(* IEC 61131-3 sources: SmartHomeNew/snapshots/project_clean_state_2026_04_16, 22 files *)

(* ---- CONSTANTS.dut ---- *)
TYPE
    C_MAX_HEATING_CIRCUITS : INT := 8;
    C_MAX_LIGHTING_ZONES : INT := 32;
    C_MAX_CLIMATE_ZONES : INT := 16;
    C_MAX_VENT_UNITS : INT := 8;
    C_MAX_DHW_UNITS : INT := 4;
    C_MAX_IO_MODULES : INT := 16;
END_TYPE

(* ---- ST_Blinds_Command_V2.dut ---- *)
TYPE ST_Blinds_Command_V2 :
STRUCT
    Position_Setpoint : BYTE;
END_STRUCT
END_TYPE

(* ---- ST_Blinds_State_V2.dut ---- *)
TYPE ST_Blinds_State_V2 :
STRUCT
    Position_Actual : BYTE;
END_STRUCT
END_TYPE

(* ---- ST_Debug_Logger_Config.dut ---- *)
{attribute 'pack_mode' := '1'}
TYPE ST_Debug_Logger_Config :
STRUCT
    enabled : BOOL;
    sampling_period_ms : UDINT := GVL_CONSTANTS.C_MS_IN_SECOND;
END_STRUCT
END_TYPE

(* ---- ST_DHW_Command_V2.dut ---- *)
TYPE ST_DHW_Command_V2 :
STRUCT
    Pump_Enable : REAL;
END_STRUCT
END_TYPE

(* ---- ST_Lifetime_Status.dut ---- *)
{attribute 'pack_mode' := '1'}
TYPE ST_Lifetime_Status :
STRUCT
    device_id : BYTE;
    runtime_hours : UDINT;
    start_count : UDINT;
    remaining_hours : UDINT;
    remaining_percent : BYTE;
    maintenance_required : BOOL;
    last_calc_timestamp : UDINT;
END_STRUCT
END_TYPE

(* ---- ST_Trend_History_Record.dut ---- *)
{attribute 'pack_mode' := '1'}
TYPE ST_Trend_History_Record :
STRUCT
    timestamp_ms : UDINT := 0;
    value : REAL := 0.0;
END_STRUCT
END_TYPE

(* ---- ST_Ventilation_State_V2.dut ---- *)
TYPE ST_Ventilation_State_V2 : STRUCT
    Supply_Temp : REAL;
END_STRUCT
END_TYPE

(* ---- FB_DHW_V2_Staging.st ---- *)
FUNCTION_BLOCK FB_DHW_V2_Staging
VAR_INPUT
    VI_Tank_ID : INT;
    VI_Enable : BOOL;
    VI_Target_Temp : REAL;
    VI_Pump_Enable : BOOL;
    VI_Heating_Priority : BOOL;
    VI_Is_Active : BOOL;
    VI_Tank_Temp : REAL;
    VI_Supply_Temp : REAL;
    VI_Return_Temp : REAL;
    VI_Pump_Actual : BOOL;
    VI_Alarm_Active : BOOL;
END_VAR
VAR_OUTPUT
    VO_Command_Shadow : ST_DHW_Command_V2;
    VO_State_Shadow : ST_DHW_State_V2;
END_VAR

IF VI_Pump_Enable THEN
    VO_Command_Shadow.Pump_Enable := 1.0;
ELSE
    VO_Command_Shadow.Pump_Enable := 0.0;
END_IF;

VO_State_Shadow.Tank_Temp := VI_Tank_Temp;
VO_State_Shadow.Supply_Temp := VI_Supply_Temp;
END_FUNCTION_BLOCK

(* ---- FB_NVRAM_Manager.st ---- *)
FUNCTION_BLOCK FB_NVRAM_Manager
VAR_INPUT
    VI_Command                  : BYTE; // 1=WRITE, 2=READ
    VI_Offset                   : UDINT; // Смещение в байтах
    VI_DataRef                  : REFERENCE TO BYTE;
    VI_DataSize                 : UDINT; // КРИТИЧНО: используем этот размер вместо SIZEOF
    VI_System_Time_MS           : UDINT;
    VI_Operator_ID              : STRING(10);
    VI_IsActivePLC              : BOOL;
    VI_TwoPersonConfirmation    : BOOL;
END_VAR
VAR_OUTPUT
    VO_Done                     : BOOL;
    VO_Error                    : BOOL;
    VO_ErrorID                  : UDINT;
    // VO_ReadDataRef removed (REFERENCE TO not allowed in output)
    VO_HMI_Status_Message       : STRING(200);
END_VAR
VAR
    L_prev_Command              : BYTE;
    L_cmd_rising                : BOOL;
    L_i                         : UDINT;
    L_Last_Write_Time_MS        : UDINT := 0; // Время последней записи
    L_Data_Changed              : BOOL; // Флаг изменения данных
    L_pData                      : POINTER TO BYTE;
END_VAR
VAR CONSTANT
    C_MAX_NVRAM_SIZE            : UDINT := 12800;
END_VAR

// Детекция фронта команды
L_cmd_rising := (VI_Command <> 0) AND (L_prev_Command = 0);
L_prev_Command := VI_Command;

IF L_cmd_rising THEN
    VO_Done := FALSE;
    VO_Error := FALSE;
    VO_ErrorID := 0;
    VO_HMI_Status_Message := '';

    // Валидация смещения
    IF VI_Offset >= C_MAX_NVRAM_SIZE THEN
        VO_Error := TRUE;
        VO_ErrorID := 16#1501;
        VO_HMI_Status_Message := 'NVRAM: Неверное смещение';
        VO_Done := TRUE;
        RETURN;
    END_IF;

    // Валидация указателя
    IF NOT __ISVALIDREF(VI_DataRef) THEN
        VO_Error := TRUE;
        VO_ErrorID := 16#150A;
        VO_HMI_Status_Message := 'NVRAM: Недействительная ссылка на данные';
        VO_Done := TRUE;
        RETURN;
    END_IF;

    L_pData := ADR(VI_DataRef);

    IF (VI_Offset + VI_DataSize) > C_MAX_NVRAM_SIZE THEN
        VO_Error := TRUE;
        VO_ErrorID := 16#150B;
        VO_HMI_Status_Message := 'NVRAM: Размер данных превышает доступный объем';
        VO_Done := TRUE;
        RETURN;
    END_IF;

    IF VI_Command = 1 THEN // ЗАПИСЬ (WRITE)
        IF NOT VI_IsActivePLC THEN
            VO_Error := TRUE;
            VO_ErrorID := 16#1509;
            VO_HMI_Status_Message := 'NVRAM: Запись запрещена (STANDBY)';
        ELSE
            // Ограничение частоты записи (не чаще 1 раза в 60 секунд)
            IF (VI_System_Time_MS - L_Last_Write_Time_MS) < 60000 AND L_Last_Write_Time_MS <> 0 THEN
                VO_Error := TRUE;
                VO_ErrorID := 16#150C;
                VO_HMI_Status_Message := 'NVRAM: Превышена частота записи (лимит 1 раз в 60с)';
            ELSE
                // Проверка на изменение данных перед записью
                L_Data_Changed := FALSE;
                IF TRUE THEN
                    L_Data_Changed := TRUE;
                END_IF;

                IF L_Data_Changed THEN
                    // Безопасное копирование (WRITE)
                    FOR L_i := 0 TO VI_DataSize - 1 DO
                        GVL_Retain.G_NVRAM_Data[VI_Offset + L_i] := L_pData[L_i];
                    END_FOR;
                    L_Last_Write_Time_MS := VI_System_Time_MS;
                    VO_HMI_Status_Message := 'NVRAM: Данные успешно сохранены в RETAIN';
                ELSE
                    VO_HMI_Status_Message := 'NVRAM: Данные не изменились, запись пропущена';
                END_IF;
            END_IF;
        END_IF;
        VO_Done := TRUE;

    ELSIF VI_Command = 2 THEN // ЧТЕНИЕ (READ)
        // Безопасное копирование (READ)
        FOR L_i := 0 TO VI_DataSize - 1 DO
            L_pData[L_i] := GVL_Retain.G_NVRAM_Data[VI_Offset + L_i];
        END_FOR;
        VO_HMI_Status_Message := 'NVRAM: Данные успешно прочитаны из RETAIN';
        VO_Done := TRUE;
    END_IF;
END_IF;

IF VI_Command = 0 THEN
    VO_Done := FALSE;
END_IF;
// >>> BULK_SYNC_ANCHOR: FB_NVRAM_Manager <<<

(* ---- FB_PID_Controller.st ---- *)
FUNCTION_BLOCK FB_PID_Controller
VAR_INPUT
    VI_SetPoint : REAL;         // Уставка
    VI_ProcessValue : REAL;     // Текущее значение
    VI_Kp : REAL;               // Коэффициент усиления
    VI_Tn : REAL;               // Время интегрирования (сек)
    VI_Tv : REAL;               // Время дифференцирования (сек)
    VI_Y_Min : REAL := 0.0;     // Минимальный выход
    VI_Y_Max : REAL := 100.0;   // Максимальный выход
    VI_Manual_Mode : BOOL;      // Ручной режим
    VI_Manual_Value : REAL;     // Значение в ручном режиме
    VI_Deadband : REAL := 0.1;  // Мертвая зона
    VI_Cycle_Time_S : REAL := 0.01; // Время цикла задачи в секундах
    VI_Reset : BOOL;            // Сброс интегральной составляющей
END_VAR
VAR_OUTPUT
    VO_Output : REAL;           // Выход регулятора
    VO_Error : REAL;            // Ошибка рассогласования
    VO_Limiting : BOOL;         // Флаг ограничения выхода (Anti-windup)
END_VAR
VAR
    L_Integral_Sum : REAL;      // Интегральная сумма
    L_Prev_Error : REAL;        // Предыдущая ошибка
    L_Derivative : REAL;        // Дифференциальная составляющая
    L_Output_Raw : REAL;        // Сырой выход до ограничения
END_VAR

// Расчет ошибки
VO_Error := VI_SetPoint - VI_ProcessValue;

// Проверка мертвой зоны
IF ABS(VO_Error) < VI_Deadband THEN
    VO_Error := 0.0;
END_IF;

IF VI_Reset THEN
    L_Integral_Sum := 0.0;
    L_Prev_Error := 0.0;
    VO_Output := 0.0;
    RETURN;
END_IF;

IF VI_Manual_Mode THEN
    VO_Output := VI_Manual_Value;
    // Безударный переход: при выходе из ручного режима выход должен остаться прежним.
    // Так как Выход = P + I + D, то I = Выход - P - D.
    // Для простоты D при переходе обнуляем (или игнорируем), тогда I = Выход - P.
    L_Integral_Sum := VO_Output - (VI_Kp * VO_Error);
    L_Prev_Error := VO_Error;
    RETURN;
END_IF;

// Пропорциональная составляющая
L_Output_Raw := VI_Kp * VO_Error;

// Интегральная составляющая (Метод трапеций)
IF VI_Tn > 0.0 THEN
    // Anti-windup: не накапливаем интеграл, если выход уже на пределе и ошибка того же знака
    IF NOT VO_Limiting OR (VO_Error > 0.0 AND L_Output_Raw < VI_Y_Max) OR (VO_Error < 0.0 AND L_Output_Raw > VI_Y_Min) THEN
        L_Integral_Sum := L_Integral_Sum + (VI_Kp / VI_Tn) * VO_Error * VI_Cycle_Time_S;
    END_IF;
    L_Output_Raw := L_Output_Raw + L_Integral_Sum;
END_IF;

// Дифференциальная составляющая
IF VI_Tv > 0.0 THEN
    L_Derivative := (VO_Error - L_Prev_Error) / VI_Cycle_Time_S;
    L_Output_Raw := L_Output_Raw + VI_Kp * VI_Tv * L_Derivative;
END_IF;

L_Prev_Error := VO_Error;

// Ограничение выхода
IF L_Output_Raw > VI_Y_Max THEN
    VO_Output := VI_Y_Max;
    VO_Limiting := TRUE;
ELSIF L_Output_Raw < VI_Y_Min THEN
    VO_Output := VI_Y_Min;
    VO_Limiting := TRUE;
ELSE
    VO_Output := L_Output_Raw;
    VO_Limiting := FALSE;
END_IF;
// >>> BULK_SYNC_ANCHOR: FB_PID_Controller <<<

(* ---- FB_Pre_Departure_Heating.st ---- *)
FUNCTION_BLOCK FB_Pre_Departure_Heating
VAR_INPUT
    VI_Departure_Time : UDINT;
    VI_System_Time    : UDINT;
END_VAR
VAR_IN_OUT
    VI_Selected       : ARRAY[1..GVL_CONSTANTS.C_MAX_HEATING_CIRCUITS] OF BOOL;
END_VAR
VAR_OUTPUT
    VO_Heating_Active : BOOL;
    VO_Setpoints      : ARRAY[1..GVL_CONSTANTS.C_MAX_HEATING_CIRCUITS] OF REAL;
END_VAR

VAR
    L_i : INT;
END_VAR

// Запуск за 3 часа (10800000 мс)
IF (SEL(VI_Departure_Time >= VI_System_Time, VI_Departure_Time - VI_System_Time, (4294967295 - VI_System_Time) + VI_Departure_Time + 1)) < 10800000 THEN
    VO_Heating_Active := TRUE;
    FOR L_i := 1 TO GVL_CONSTANTS.C_MAX_HEATING_CIRCUITS DO
        IF VI_Selected[L_i] THEN VO_Setpoints[L_i] := 22.0; END_IF;
    END_FOR;
ELSE
    VO_Heating_Active := FALSE;
END_IF;

(* ---- FB_Presence_Playback.st ---- *)
FUNCTION_BLOCK FB_Presence_Playback
VAR_INPUT
    VI_Mode_Record : BOOL; // TRUE - записываем, FALSE - воспроизводим
    VI_Time_Index   : UDINT; // Индекс времени в рамках недели (мс)
END_VAR
VAR_IN_OUT
    VI_Light_Inputs : ARRAY[1..32] OF BOOL;
END_VAR
VAR_OUTPUT
    VO_Light_Outputs : ARRAY[1..32] OF BOOL;
END_VAR
VAR
    L_Current_Slot : UDINT;
    L_i : INT;
END_VAR

L_Current_Slot := (VI_Time_Index / (GVL_CONSTANTS.C_MS_IN_MINUTE * 10)) MOD TO_UDINT(GVL_CONSTANTS.C_MAX_PRESENCE_HISTORY); // Слот каждые 10 минут

IF VI_Mode_Record THEN
    // Запись текущего состояния в слот
    GVL_Retain.G_Presence_History[L_Current_Slot] := 0;
    FOR L_i := 1 TO 32 DO
        IF VI_Light_Inputs[L_i] THEN
            GVL_Retain.G_Presence_History[L_Current_Slot] := GVL_Retain.G_Presence_History[L_Current_Slot] OR SHL(WORD#1, L_i-1);
        END_IF;
    END_FOR;
ELSE
    // Воспроизведение из слота
    FOR L_i := 1 TO 32 DO
        VO_Light_Outputs[L_i] := (GVL_Retain.G_Presence_History[L_Current_Slot] AND SHL(WORD#1, L_i-1)) <> 0;
    END_FOR;
END_IF;

(* ---- FB_Redundancy_Manager.st ---- *)
FUNCTION_BLOCK FB_Redundancy_Manager
VAR_INPUT
    VI_System_Time_MS : UDINT; // Системное время (мс)
    VI_Local_PLC_ID : BYTE; // 1 = ПЛК А, 2 = ПЛК B
    VI_Remote_Pulse : BOOL; // Сигнал от партнера
    VI_Remote_Is_Active : BOOL; // Статус партнера
    VI_Gateway_Ping_OK : BOOL; // Пинг до шлюза
    VI_Remote_State : ST_System_State_Snapshot; // Состояние партнера
    VI_Local_State : ST_System_State_Snapshot; // Локальное состояние
END_VAR
VAR_OUTPUT
    VO_Local_Role : E_PLC_ROLE; // Локальная роль ПЛК (Active/Standby)
    VO_Local_Pulse : BOOL; // Локальный сигнал пульса для партнера
    VO_Sync_Data_Req : BOOL; // Запрос на синхронизацию данных
    VO_Status_Msg : STRING(200); // Строковое сообщение о статусе
    VO_Synced_State : ST_System_State_Snapshot; // Синхронизированное состояние
    VO_State_Updated : BOOL; // Флаг: Состояние было обновлено
END_VAR
VAR
    L_Heartbeat : FB_PLC_Heartbeat;
    L_Pulse_Timer : FB_System_Timer;
    L_Pulse_State : BOOL;
    L_Prev_Role : E_PLC_ROLE;
    L_State_Replicator : FB_State_Replication;
END_VAR

// 1. Генерация собственного пульса (меандр 100 мс)
L_Pulse_Timer(IN := NOT L_Pulse_Timer.Q, PT := T#100ms, VI_System_Time_MS := VI_System_Time_MS);
IF L_Pulse_Timer.Q THEN
    L_Pulse_State := NOT L_Pulse_State;
END_IF;
VO_Local_Pulse := L_Pulse_State;

// 2. Определение роли через Heartbeat
L_Heartbeat(
    VI_Local_ID := VI_Local_PLC_ID,
    VI_System_Time := VI_System_Time_MS,
    VI_Remote_Pulse := VI_Remote_Pulse,
    VI_Remote_Is_Active := VI_Remote_Is_Active,
    VI_Gateway_Ping_OK := VI_Gateway_Ping_OK
);

IF L_Heartbeat.VO_Is_Active THEN
    VO_Local_Role := E_PLC_ROLE.ROLE_ACTIVE;
    VO_Status_Msg := 'ПЛК АКТИВЕН (ВЕДУЩИЙ)';
ELSE
    VO_Local_Role := E_PLC_ROLE.ROLE_STANDBY;
    VO_Status_Msg := 'ПЛК В РЕЗЕРВЕ (ВЕДОМЫЙ)';
END_IF;

// 3. Запрос на синхронизацию при переходе в ACTIVE
IF VO_Local_Role = E_PLC_ROLE.ROLE_ACTIVE AND L_Prev_Role = E_PLC_ROLE.ROLE_STANDBY THEN
    VO_Sync_Data_Req := TRUE;
ELSE
    VO_Sync_Data_Req := FALSE;
END_IF;

L_State_Replicator(
    VI_Local_Role := VO_Local_Role,
    VI_Sync_Req := VO_Sync_Data_Req,
    VI_Local_State := VI_Local_State,
    VI_Remote_State := VI_Remote_State,
    VI_System_Time_MS := VI_System_Time_MS
);
VO_Synced_State := L_State_Replicator.VO_Synced_State;
VO_State_Updated := L_State_Replicator.VO_State_Updated;

L_Prev_Role := VO_Local_Role;
// >>> BULK_SYNC_ANCHOR: FB_Redundancy_Manager <<<

(* ---- FB_Rule_Engine.st ---- *)
FUNCTION_BLOCK FB_Rule_Engine
VAR_INPUT
    VI_System_Time_MS : UDINT; // Системное время (мс)
    VI_IsActivePLC : BOOL; // Флаг: Данный ПЛК является ведущим
    VI_Security_Armed : BOOL; // Статус: Система под охраной
    VI_Current_Time : TOD; // Текущее время суток
    VI_Day_Of_Week : INT; // Текущий день недели (1..7, 1 = Понедельник)
END_VAR
VAR_IN_OUT
    VI_Rules : ARRAY[1..GVL_CONSTANTS.C_MAX_RULES] OF ST_User_Rule; // Массив пользовательских правил
    VI_Indoor_Temps : ARRAY[1..16] OF REAL; // Температуры в помещениях
    VI_Floor_Temps : ARRAY[1..8] OF REAL; // Температуры пола
    VI_Humidities : ARRAY[1..16] OF REAL; // Влажность в помещениях
    VI_CO2_Levels : ARRAY[1..16] OF REAL; // Уровни CO2
    VI_Motion_Sensors : ARRAY[1..16] OF BOOL; // Датчики движения
    VI_Door_Sensors : ARRAY[1..GVL_CONSTANTS.C_MAX_DOOR_SENSORS] OF BOOL; // Датчики открытия дверей
    VI_Window_Sensors : ARRAY[1..16] OF BOOL; // Датчики открытия окон
    VI_Water_Sensors : ARRAY[1..GVL_CONSTANTS.C_MAX_FLOOD_SENSORS] OF BOOL; // Датчики протечки воды
    VI_Smoke_Sensors : ARRAY[1..GVL_CONSTANTS.C_MAX_SMOKE_SENSORS] OF BOOL; // Датчики дыма
    VI_Methane_Sensors : ARRAY[1..GVL_CONSTANTS.C_MAX_METHANE_SENSORS] OF REAL; // Датчики метана
    VI_CO_Sensors : ARRAY[1..GVL_CONSTANTS.C_MAX_CO_SENSORS] OF REAL; // Датчики угарного газа
END_VAR
VAR_OUTPUT
    VO_Actions : ARRAY[1..GVL_CONSTANTS.C_MAX_RULES] OF ST_Rule_Action; // Сформированные действия по правилам
END_VAR
VAR
    L_i : INT;
    fbCompat : ARRAY[1..GVL_CONSTANTS.C_MAX_RULES] OF FB_Rule_Compatibility_Package;
    L_Compat_All_OK : BOOL;
    L_Compat_First_Warning : STRING(255);
    L_Compat_First_Warning_Latched : BOOL;
    L_Shadow_V2_Enabled : BOOL;
    L_Shadow_V2_Roundtrip_Mismatch : BOOL;
    L_Shadow_V2_First_Mismatch_Rule : INT;
    L_V2_Switch_Enabled : BOOL;
    L_V2_Path_Ready : BOOL;
    L_V2_Using_Legacy_Fallback : BOOL;
    L_Condition_Met : BOOL;
    L_Current_Value : REAL;
    L_Triggers : ARRAY[1..GVL_CONSTANTS.C_MAX_RULES] OF R_TRIG;
    L_Trigger_Count : ARRAY[1..GVL_CONSTANTS.C_MAX_RULES] OF UINT;
    L_Last_Reset_Time : UDINT;
    L_Elapsed_Time : UDINT;
END_VAR

IF NOT VI_IsActivePLC THEN RETURN; END_IF;

L_Compat_All_OK := TRUE;
L_Compat_First_Warning := '';
L_Compat_First_Warning_Latched := FALSE;
L_Shadow_V2_Enabled := TRUE;
L_Shadow_V2_Roundtrip_Mismatch := FALSE;
L_Shadow_V2_First_Mismatch_Rule := 0;
L_V2_Switch_Enabled := FALSE;
L_V2_Path_Ready := FALSE;
L_V2_Using_Legacy_Fallback := TRUE;

// Сброс счетчиков срабатываний каждую минуту (защита от циклических зависимостей/дребезга)
L_Elapsed_Time := (SEL(VI_System_Time_MS >= L_Last_Reset_Time, VI_System_Time_MS - L_Last_Reset_Time, (4294967295 - L_Last_Reset_Time) + VI_System_Time_MS + 1));

IF L_Elapsed_Time >= GVL_CONSTANTS.C_MS_IN_MINUTE THEN
    L_Last_Reset_Time := VI_System_Time_MS;
    FOR L_i := 1 TO GVL_CONSTANTS.C_MAX_RULES DO
        L_Trigger_Count[L_i] := 0;
    END_FOR;
END_IF;

FOR L_i := 1 TO GVL_CONSTANTS.C_MAX_RULES DO
    fbCompat[L_i](VI_Rule_Legacy := VI_Rules[L_i]);

    IF NOT fbCompat[L_i].VO_Forward_OK OR NOT fbCompat[L_i].VO_Reverse_OK THEN
        L_Compat_All_OK := FALSE;
    END_IF;

    IF (NOT L_Compat_First_Warning_Latched) AND (fbCompat[L_i].VO_Warning_Text <> '') THEN
        L_Compat_First_Warning := fbCompat[L_i].VO_Warning_Text;
        L_Compat_First_Warning_Latched := TRUE;
    END_IF;

    IF L_Shadow_V2_Enabled THEN
        IF (fbCompat[L_i].VO_Rule_Legacy_Roundtrip.Action_Type <> VI_Rules[L_i].Action_Type)
           OR (fbCompat[L_i].VO_Rule_Legacy_Roundtrip.Action_Target_ID <> VI_Rules[L_i].Action_Target_ID)
           OR (ABS(fbCompat[L_i].VO_Rule_Legacy_Roundtrip.Action_Value - VI_Rules[L_i].Action_Value) > 0.0001)
           OR (fbCompat[L_i].VO_Rule_Legacy_Roundtrip.Condition_Type <> VI_Rules[L_i].Condition_Type)
           OR (fbCompat[L_i].VO_Rule_Legacy_Roundtrip.Condition_Target_ID <> VI_Rules[L_i].Condition_Target_ID)
           OR (fbCompat[L_i].VO_Rule_Legacy_Roundtrip.Condition_Op <> VI_Rules[L_i].Condition_Op)
           OR (ABS(fbCompat[L_i].VO_Rule_Legacy_Roundtrip.Condition_Value - VI_Rules[L_i].Condition_Value) > 0.0001)
           OR (ABS(fbCompat[L_i].VO_Rule_Legacy_Roundtrip.Condition_Value_Max - VI_Rules[L_i].Condition_Value_Max) > 0.0001) THEN
            L_Shadow_V2_Roundtrip_Mismatch := TRUE;
            IF L_Shadow_V2_First_Mismatch_Rule = 0 THEN
                L_Shadow_V2_First_Mismatch_Rule := L_i;
            END_IF;
        END_IF;
    END_IF;

    // Phase 4 scaffold: optional V2 switch point.
    // Current state: always remain on legacy behavior.
    // Future state: when V2 path is implemented and validated,
    // this block becomes the controlled branch point.
    IF L_V2_Switch_Enabled AND L_V2_Path_Ready THEN
        L_V2_Using_Legacy_Fallback := FALSE;
        // V2 action-generation path placeholder.
        // No runtime behavior change yet.
    ELSE
        L_V2_Using_Legacy_Fallback := TRUE;
    END_IF;

    VO_Actions[L_i].Active := FALSE;
    IF VI_Rules[L_i].Enabled THEN
        L_Condition_Met := FALSE;
        L_Current_Value := 0.0;

        // Определение значения для проверки
        IF VI_Rules[L_i].Condition_Target_ID > 0 THEN
            CASE VI_Rules[L_i].Condition_Type OF
                E_Rule_Condition_Type.COND_AIR_TEMP: IF VI_Rules[L_i].Condition_Target_ID <= 16 THEN L_Current_Value := VI_Indoor_Temps[VI_Rules[L_i].Condition_Target_ID]; END_IF;
                E_Rule_Condition_Type.COND_FLOOR_TEMP: IF VI_Rules[L_i].Condition_Target_ID <= 8 THEN L_Current_Value := VI_Floor_Temps[VI_Rules[L_i].Condition_Target_ID]; END_IF;
                E_Rule_Condition_Type.COND_HUMIDITY: IF VI_Rules[L_i].Condition_Target_ID <= 16 THEN L_Current_Value := VI_Humidities[VI_Rules[L_i].Condition_Target_ID]; END_IF;
                E_Rule_Condition_Type.COND_CO2: IF VI_Rules[L_i].Condition_Target_ID <= 16 THEN L_Current_Value := VI_CO2_Levels[VI_Rules[L_i].Condition_Target_ID]; END_IF;
                E_Rule_Condition_Type.COND_MOTION: IF VI_Rules[L_i].Condition_Target_ID <= 16 THEN L_Current_Value := SEL(VI_Motion_Sensors[VI_Rules[L_i].Condition_Target_ID], 0.0, 1.0); END_IF;
                E_Rule_Condition_Type.COND_DOOR_WINDOW:
                    IF VI_Rules[L_i].Condition_Target_ID <= GVL_CONSTANTS.C_MAX_DOOR_SENSORS THEN
                        L_Current_Value := SEL(VI_Door_Sensors[VI_Rules[L_i].Condition_Target_ID] OR VI_Window_Sensors[VI_Rules[L_i].Condition_Target_ID], 0.0, 1.0);
                    ELSIF VI_Rules[L_i].Condition_Target_ID <= 16 THEN
                        L_Current_Value := SEL(VI_Window_Sensors[VI_Rules[L_i].Condition_Target_ID], 0.0, 1.0);
                    END_IF;
                E_Rule_Condition_Type.COND_FLOOD: IF VI_Rules[L_i].Condition_Target_ID <= GVL_CONSTANTS.C_MAX_FLOOD_SENSORS THEN L_Current_Value := SEL(VI_Water_Sensors[VI_Rules[L_i].Condition_Target_ID], 0.0, 1.0); END_IF;
                E_Rule_Condition_Type.COND_SMOKE: IF VI_Rules[L_i].Condition_Target_ID <= GVL_CONSTANTS.C_MAX_SMOKE_SENSORS THEN L_Current_Value := SEL(VI_Smoke_Sensors[VI_Rules[L_i].Condition_Target_ID], 0.0, 1.0); END_IF;
                E_Rule_Condition_Type.COND_METHANE: IF VI_Rules[L_i].Condition_Target_ID <= GVL_CONSTANTS.C_MAX_METHANE_SENSORS THEN L_Current_Value := VI_Methane_Sensors[VI_Rules[L_i].Condition_Target_ID]; END_IF;
                E_Rule_Condition_Type.COND_CO: IF VI_Rules[L_i].Condition_Target_ID <= GVL_CONSTANTS.C_MAX_CO_SENSORS THEN L_Current_Value := VI_CO_Sensors[VI_Rules[L_i].Condition_Target_ID]; END_IF;
                E_Rule_Condition_Type.COND_TIME_OF_DAY: L_Current_Value := TO_REAL(TOD_TO_UDINT(VI_Current_Time) / GVL_CONSTANTS.C_MS_IN_MINUTE); // Время в минутах
                E_Rule_Condition_Type.COND_DAY_OF_WEEK: L_Current_Value := TO_REAL(VI_Day_Of_Week);
            END_CASE;
        ELSE
            IF VI_Rules[L_i].Condition_Type = E_Rule_Condition_Type.COND_TIME_OF_DAY THEN
                L_Current_Value := TO_REAL(TOD_TO_UDINT(VI_Current_Time) / GVL_CONSTANTS.C_MS_IN_MINUTE); // Время в минутах
            ELSIF VI_Rules[L_i].Condition_Type = E_Rule_Condition_Type.COND_DAY_OF_WEEK THEN
                L_Current_Value := TO_REAL(VI_Day_Of_Week);
            END_IF;
        END_IF;

        // Проверка условия
        CASE VI_Rules[L_i].Condition_Op OF
            E_Rule_Comparison.COMP_GT: L_Condition_Met := (L_Current_Value > VI_Rules[L_i].Condition_Value);
            E_Rule_Comparison.COMP_LT: L_Condition_Met := (L_Current_Value < VI_Rules[L_i].Condition_Value);
            E_Rule_Comparison.COMP_EQ: L_Condition_Met := (ABS(L_Current_Value - VI_Rules[L_i].Condition_Value) < 0.1);
            E_Rule_Comparison.COMP_GE: L_Condition_Met := (L_Current_Value >= VI_Rules[L_i].Condition_Value);
            E_Rule_Comparison.COMP_LE: L_Condition_Met := (L_Current_Value <= VI_Rules[L_i].Condition_Value);
            E_Rule_Comparison.COMP_IN_RANGE: L_Condition_Met := (L_Current_Value >= VI_Rules[L_i].Condition_Value) AND (L_Current_Value <= VI_Rules[L_i].Condition_Value_Max);
            E_Rule_Comparison.COMP_TRUE: L_Condition_Met := (L_Current_Value > 0.5);
            E_Rule_Comparison.COMP_FALSE: L_Condition_Met := (L_Current_Value < 0.5);
        END_CASE;

        // Формирование действия
        L_Triggers[L_i](CLK := L_Condition_Met);

        IF L_Triggers[L_i].Q THEN
            L_Trigger_Count[L_i] := L_Trigger_Count[L_i] + 1;
            IF L_Trigger_Count[L_i] > 10 THEN
                // ТЗ 13.5: Блокировка правила при слишком частом срабатывании (циклическая зависимость)
                VO_Actions[L_i].Active := FALSE;
                VO_Actions[L_i].Triggered := FALSE;
                CONTINUE; // Пропускаем выполнение
            END_IF;
        END_IF;

        IF L_Condition_Met AND (L_Trigger_Count[L_i] <= 10) THEN
            VO_Actions[L_i].Active := TRUE;
            VO_Actions[L_i].Triggered := L_Triggers[L_i].Q;
            VO_Actions[L_i].Action_Type := VI_Rules[L_i].Action_Type;
            VO_Actions[L_i].Target_ID := VI_Rules[L_i].Action_Target_ID;
            VO_Actions[L_i].Value := VI_Rules[L_i].Action_Value;
        END_IF;
    END_IF;
END_FOR;
// >>> BULK_SYNC_ANCHOR: FB_Rule_Engine <<<

(* ---- FB_State_Manager_MVP.st ---- *)
FUNCTION_BLOCK FB_State_Manager
VAR_INPUT
    VI_Gas_Alarm     : BOOL;
    VI_Fire_Alarm    : BOOL;
    VI_Flood_Alarm   : BOOL;

    VI_IO_Healthy    : BOOL;
    VI_Freeze_Risk   : BOOL;

    VI_Reset_Request : BOOL;
END_VAR

VAR_OUTPUT
    VO_System_Mode : INT; // temporary, replace with ENUM later
END_VAR

VAR
    L_Fire_Latched  : BOOL;
    L_Gas_Latched   : BOOL;
    L_Flood_Latched : BOOL;
END_VAR

// Fire latch
IF VI_Fire_Alarm THEN
    L_Fire_Latched := TRUE;
END_IF;
IF VI_Reset_Request AND NOT VI_Fire_Alarm THEN
    L_Fire_Latched := FALSE;
END_IF;

// Gas latch
IF VI_Gas_Alarm THEN
    L_Gas_Latched := TRUE;
END_IF;
IF VI_Reset_Request AND NOT VI_Gas_Alarm THEN
    L_Gas_Latched := FALSE;
END_IF;

// Flood latch
IF VI_Flood_Alarm THEN
    L_Flood_Latched := TRUE;
END_IF;
IF VI_Reset_Request AND NOT VI_Flood_Alarm THEN
    L_Flood_Latched := FALSE;
END_IF;

// Mode logic
IF L_Fire_Latched THEN
    VO_System_Mode := 2; // SAFE_STOP
ELSIF L_Flood_Latched THEN
    VO_System_Mode := 2;
ELSIF L_Gas_Latched THEN
    IF VI_Freeze_Risk THEN
        VO_System_Mode := 3; // FREEZE
    ELSE
        VO_System_Mode := 1; // DEGRADED
    END_IF;
ELSIF NOT VI_IO_Healthy THEN
    VO_System_Mode := 1;
ELSE
    VO_System_Mode := 0; // NORMAL
END_IF;

(* ---- FB_State_Snapshot_NVRAM.st ---- *)
FUNCTION_BLOCK FB_State_Snapshot_NVRAM
VAR_INPUT
    VI_System_Time_MS : UDINT;
    VI_Save_Req       : BOOL;
    VI_Snapshot       : ST_State_Snapshot;
END_VAR
VAR_OUTPUT
    VO_Saved          : BOOL;
    VO_Error          : BOOL;
END_VAR
VAR
    L_FileName        : STRING := '/home/root/snapshot.bin';
    L_State           : INT := 0;

    // Асинхронные блоки из библиотеки CAA_File
    fbFileOpen        : FILE.Open;
    fbFileWrite       : FILE.Write;
    fbFileClose       : FILE.Close;
    L_FileHandle      : FILE.HANDLE;
END_VAR

CASE L_State OF
    0: // Ожидание
        VO_Saved := FALSE;
        VO_Error := FALSE;
        IF VI_Save_Req THEN
            L_State := 10;
            fbFileOpen(xExecute := FALSE);
            fbFileWrite(xExecute := FALSE);
            fbFileClose(xExecute := FALSE);
        END_IF;

    10: // Открытие файла
        fbFileOpen(
            xExecute := TRUE,
            sFileName := L_FileName,
            eFileMode := FILE.MODE.MWRITE
        );
        IF fbFileOpen.xDone THEN
            L_FileHandle := fbFileOpen.hFile;
            fbFileOpen(xExecute := FALSE);
            L_State := 20;
        ELSIF fbFileOpen.xError THEN
            VO_Error := TRUE;
            L_State := 0;
        END_IF;

    20: // Запись
        fbFileWrite(
            xExecute := TRUE,
            hFile := L_FileHandle,
            pBuffer := ADR(VI_Snapshot),
            szSize := SIZEOF(VI_Snapshot)
        );
        IF fbFileWrite.xDone THEN
            fbFileWrite(xExecute := FALSE);
            L_State := 30;
        ELSIF fbFileWrite.xError THEN
            VO_Error := TRUE;
            L_State := 30; // Все равно закрываем файл
        END_IF;

    30: // Закрытие
        fbFileClose(
            xExecute := TRUE,
            hFile := L_FileHandle
        );
        IF fbFileClose.xDone THEN
            fbFileClose(xExecute := FALSE);
            IF NOT VO_Error THEN
                VO_Saved := TRUE;
            END_IF;
            L_State := 0;
        ELSIF fbFileClose.xError THEN
            VO_Error := TRUE;
            L_State := 0;
        END_IF;
END_CASE;

(* ---- FB_Supply_Ventilation_Controller.st ---- *)
FUNCTION_BLOCK FB_Supply_Ventilation_Controller
VAR_INPUT
    VI_Outdoor_Temp : REAL;
    VI_Supply_Temp  : REAL; // Температура приточного воздуха
    VI_Target_Temp  : REAL;
    VI_Config       : ST_Ventilation_Unit_Config;
END_VAR
VAR_OUTPUT
    VO_Heater_Power : REAL; // 0-100%
    VO_Fan_Speed    : BYTE; // 0-100%
END_VAR
VAR
    L_PID : FB_PID_Controller;
END_VAR

// ПИД-регулятор калорифера
L_PID(
    VI_SetPoint := VI_Target_Temp,
    VI_ProcessValue := VI_Supply_Temp, // Используем датчик притока
    VI_Kp := 5.0, VI_Tn := 60.0, VI_Tv := 0.0,
    VI_Y_Min := 0.0, VI_Y_Max := 100.0, VI_Cycle_Time_S := 1.0,
    VO_Output => VO_Heater_Power
);

VO_Fan_Speed := 50; // Базовая скорость

(* ---- FB_Valve_Test.st ---- *)
FUNCTION_BLOCK FB_Valve_Test
VAR_INPUT
    VI_System_Time_MS : UDINT;
    VI_Start_Test     : BOOL;
    VI_Valve_ID       : BYTE;
END_VAR
VAR_OUTPUT
    VO_Test_Active    : BOOL;
    VO_Result         : E_Valve_Test_Result;
    VO_Valve_Cmd      : BOOL;
END_VAR
VAR
    L_Start_Time      : UDINT;
    L_State           : INT;
END_VAR

CASE L_State OF
    0: // Ожидание
        IF VI_Start_Test THEN
            VO_Test_Active := TRUE;
            VO_Result := E_Valve_Test_Result.TEST_IN_PROGRESS;
            L_Start_Time := VI_System_Time_MS;
            VO_Valve_Cmd := TRUE; // Открыть
            L_State := 1;
        END_IF;
    1: // Тест
        IF (SEL(VI_System_Time_MS >= L_Start_Time, VI_System_Time_MS - L_Start_Time, (4294967295 - L_Start_Time) + VI_System_Time_MS + 1)) > 5000 THEN
            VO_Valve_Cmd := FALSE; // Закрыть
            VO_Result := E_Valve_Test_Result.TEST_PASSED; // Заглушка, нужен контроль концевиков
            VO_Test_Active := FALSE;
            L_State := 0;
        END_IF;
END_CASE;

(* ---- FB_Valve_Test_Manager.st ---- *)
FUNCTION_BLOCK FB_Valve_Test_Manager
VAR_INPUT
    VI_System_Time_MS : UDINT;
    VI_IsActivePLC : BOOL;
END_VAR
VAR_IN_OUT
    VI_Valve_Currents : ARRAY[1..GVL_CONSTANTS.C_MAX_MANIFOLDS] OF REAL;
    VI_Valve_End_Switches : ARRAY[1..GVL_CONSTANTS.C_MAX_MANIFOLDS] OF BOOL;
    VI_Config : ARRAY[1..GVL_CONSTANTS.C_MAX_MANIFOLDS] OF ST_Valve_Test_Config;
END_VAR
VAR_OUTPUT
    VO_Test_Active : BOOL;
    VO_Current_Valve : INT; // Текущий тестируемый клапан
    VO_Valve_Cmd : ARRAY[1..GVL_CONSTANTS.C_MAX_MANIFOLDS] OF BOOL;
    VO_Test_Results : ARRAY[1..GVL_CONSTANTS.C_MAX_MANIFOLDS] OF BOOL; // TRUE = OK
    VO_Status_Msg : STRING(200);
END_VAR
VAR
    L_State : INT;
    L_Current_Valve : INT := 1;
    L_Test_Start_Time : UDINT;
    L_Last_Test_Time : ARRAY[1..GVL_CONSTANTS.C_MAX_MANIFOLDS] OF UDINT;
    L_i : INT;
    L_Need_Test : BOOL;
    L_Elapsed_Time : UDINT;
END_VAR

IF NOT VI_IsActivePLC THEN RETURN; END_IF;

CASE L_State OF
    0: // Ожидание
        VO_Test_Active := FALSE;
        L_Need_Test := FALSE;

        // Поиск клапана, которому нужен тест (раз в неделю)
        FOR L_i := 1 TO GVL_CONSTANTS.C_MAX_MANIFOLDS DO
            IF VI_Config[L_i].enabled AND ((VI_System_Time_MS - L_Last_Test_Time[L_i]) > (VI_Config[L_i].test_interval_days * 86400000)) THEN
                L_Current_Valve := L_i;
                L_Need_Test := TRUE;
                EXIT;
            END_IF;
        END_FOR;

        IF L_Need_Test THEN
            L_State := 1;
            L_Test_Start_Time := VI_System_Time_MS;
            VO_Test_Active := TRUE;
            VO_Current_Valve := L_Current_Valve;
            VO_Valve_Cmd[L_Current_Valve] := TRUE; // Открываем
            VO_Status_Msg := CONCAT('ТЕСТ КЛАПАНА ', INT_TO_STRING(L_Current_Valve));
            VO_Test_Results[L_Current_Valve] := TRUE; // Сброс результата
        END_IF;

    1: // Тестирование (ожидание открытия)
        L_Elapsed_Time := (VI_System_Time_MS - L_Test_Start_Time);

        IF VI_Valve_End_Switches[L_Current_Valve] THEN
            // Концевик сработал до истечения таймаута
            // Проверка тока
            IF ABS(VI_Valve_Currents[L_Current_Valve] - VI_Config[L_Current_Valve].Nominal_Current) > (VI_Config[L_Current_Valve].Nominal_Current * 0.2) THEN
                VO_Test_Results[L_Current_Valve] := FALSE; // Ошибка по току
            END_IF;

            GVL_Retain.G_Valve_Test_Results[L_Current_Valve] := VO_Test_Results[L_Current_Valve];

            VO_Valve_Cmd[L_Current_Valve] := FALSE; // Закрываем
            L_Test_Start_Time := VI_System_Time_MS; // Перезапускаем таймер для проверки закрытия
            L_State := 2;
        ELSIF L_Elapsed_Time > TO_UDINT(VI_Config[L_Current_Valve].nominal_close_time_sec * 1000.0) THEN
            // Таймаут открытия (заклинивание)
            VO_Test_Results[L_Current_Valve] := FALSE;
            GVL_Retain.G_Valve_Test_Results[L_Current_Valve] := FALSE;
            VO_Status_Msg := CONCAT('ОШИБКА: ЗАКЛИНИВАНИЕ КЛАПАНА ', INT_TO_STRING(L_Current_Valve));

            VO_Valve_Cmd[L_Current_Valve] := FALSE; // Закрываем
            L_Test_Start_Time := VI_System_Time_MS; // Перезапускаем таймер
            L_State := 2;
        END_IF;

    2: // Ожидание закрытия
        L_Elapsed_Time := (VI_System_Time_MS - L_Test_Start_Time);

        IF NOT VI_Valve_End_Switches[L_Current_Valve] THEN
            // Концевик разомкнулся (клапан закрыт)
            L_Last_Test_Time[L_Current_Valve] := VI_System_Time_MS;
            L_State := 0;
            IF VO_Test_Results[L_Current_Valve] THEN
                VO_Status_Msg := 'ТЕСТ ЗАВЕРШЕН УСПЕШНО';
            END_IF;
        ELSIF L_Elapsed_Time > TO_UDINT(VI_Config[L_Current_Valve].nominal_close_time_sec * 1000.0) THEN
            // Таймаут закрытия (заклинивание)
            VO_Test_Results[L_Current_Valve] := FALSE;
            GVL_Retain.G_Valve_Test_Results[L_Current_Valve] := FALSE;
            VO_Status_Msg := CONCAT('ОШИБКА: НЕ ЗАКРЫЛСЯ КЛАПАН ', INT_TO_STRING(L_Current_Valve));

            L_Last_Test_Time[L_Current_Valve] := VI_System_Time_MS;
            L_State := 0;
        END_IF;
END_CASE;

(* ---- PRG_Heating.st ---- *)
PROGRAM PRG_Heating
VAR
    fbHeatingManager : FB_Heating_System_Manager;
    fbDHWManager : FB_DHW_Manager;
    L_i : INT;
    L_Zone_Valves_8 : ARRAY[1..8] OF BOOL;
    L_Boiler_Modulation_REAL : ARRAY[1..GVL_CONSTANTS.C_MAX_BOILERS] OF REAL;
    L_Heating_Emergency_Stop : BOOL;
    L_Heating_Gas_Safety_Stop : BOOL;
    L_Heating_DHW_Demand : BOOL;
END_VAR

FOR L_i := 1 TO GVL_CONSTANTS.C_MAX_BOILERS DO
    L_Boiler_Modulation_REAL[L_i] := TO_REAL(GVL_IO.AI_Boiler_Modulation[L_i]);
END_FOR;

// === Heating Arbitration ===
L_Heating_Emergency_Stop := GVL_STATE.G_Safety_Emergency_Stop;
L_Heating_Gas_Safety_Stop := GVL_STATE.G_Safety_Gas_Latched;
L_Heating_DHW_Demand := fbDHWManager.VO_Heating_Pump;

// Priority 1: emergency stop
IF L_Heating_Emergency_Stop THEN
    L_Heating_Gas_Safety_Stop := FALSE;
    L_Heating_DHW_Demand := FALSE;
// Priority 2: gas safety stop
ELSIF L_Heating_Gas_Safety_Stop THEN
    L_Heating_DHW_Demand := FALSE;
ELSIF GVL_STATE.G_System_Mode = E_System_Operating_Mode.MODE_DEGRADED THEN
    L_Heating_DHW_Demand := FALSE;
END_IF;

// 9. Управление климатом (Отопление)
fbHeatingManager(
    VI_System_Time_MS := GVL_STATUS.G_System_Time_MS,
    VI_Current_TOD := GVL_STATUS.G_Current_TOD,
    VI_IsActivePLC := GVL_STATUS.G_Is_Active_PLC,
    VI_Outdoor_Temp := GVL_STATE.G_Outdoor_Temp,
    VI_Floor_Temps := GVL_STATE.G_Floor_Temps,
    VI_Room_Temps := GVL_STATE.G_Room_Temps,
    VI_Config := GVL_CONFIG.G_Heating_Config,
    VI_Zone_Configs := GVL_CONFIG.G_HMI_FloorHeating_Configs,
    VI_Tariff := GVL_CONFIG.G_HMI_Tariff_Settings,
    VI_Current_Hour := TO_UINT(GVL_STATUS.G_Time_Of_Day_MS / GVL_CONSTANTS.C_MS_IN_HOUR),
    VI_Manifold_Pressures := GVL_STATE.G_Manifold_Pressures,
    VI_Manifold_Currents := GVL_STATE.G_Manifold_Currents,
    VI_Manifold_Temps_Supply := GVL_STATE.G_Manifold_T_Supply,
    VI_Manifold_Temps_Return := GVL_STATE.G_Manifold_T_Return,
    VI_Boiler_Flame_Status := GVL_STATE.G_Boiler_Flame,
    VI_Boiler_Error_Status := GVL_STATE.G_Boiler_Error,
    VI_Boiler_OT_Online := GVL_STATE.G_Boiler_OT_Online,
    VI_Boiler_Modulation := L_Boiler_Modulation_REAL,
    VI_Rule_Actions := GVL_STATE.G_Rule_Actions,
    VI_Boiler_Stop := FALSE, // legacy input disabled; safety flows via mode/latches
    VI_IO_Modules_Online := GVL_STATUS.G_IO_Modules_Online,
    VI_DHW_Heating_Demand := L_Heating_DHW_Demand,
    VI_DHW_Target_Temp := GVL_CONFIG.G_DHW_Config.Target_Temp,
    VI_Current_Scenario := GVL_STATUS.G_Current_Scenario,
    VI_System_Mode := GVL_STATE.G_System_Mode,
    VI_Emergency_Stop := L_Heating_Emergency_Stop,
    VI_Gas_Safety_Stop := L_Heating_Gas_Safety_Stop,
    VI_Scenario_Configs := GVL_CONFIG.G_HMI_Scenario_Configs,
    VI_Manifold_End_Switches := GVL_STATE.G_Manifold_End_Switches,
    VI_Valve_Test_Config := GVL_CONFIG.G_Valve_Test_Config,
    VO_Manifold_Valves => GVL_STATE.G_Manifold_Valves,
    VO_Manifold_Pumps => GVL_STATE.G_Manifold_Pumps,
    VO_Zone_Valves => L_Zone_Valves_8,
    VO_Boiler_OT_Enable => GVL_STATE.G_Boiler_OT_Enable,
    VO_Boiler_OT_Setpoint => GVL_STATE.G_Boiler_OT_Setpoint,
    VO_Backup_Circulation_Pump => GVL_STATE.G_Backup_Circulation_Pump,
    VO_Electric_Heater_Enable => GVL_STATE.G_Electric_Heater_Enable,
    VO_Freeze_Risk_Status => GVL_STATE.G_Safety_Freeze_Risk,
    VO_Status => GVL_STATUS.G_Manifold_Status,
    VO_Boiler_Status => GVL_STATUS.G_Boiler_Status
);

// 12. Управление ГВС
fbDHWManager(
    VI_System_Time_MS := GVL_STATUS.G_System_Time_MS,
    VI_Current_TOD := GVL_STATUS.G_Current_TOD,
    VI_IsActivePLC := GVL_STATUS.G_Is_Active_PLC,
    VI_Temp := GVL_STATE.G_DHW_Temp,
    VI_Pressure := GVL_STATE.G_DHW_Pressure,
    VI_Config := GVL_CONFIG.G_DHW_Config,
    VI_Current_Day_Of_Week := GVL_STATUS.G_Current_Day,
    VI_IO_Modules_Online := GVL_STATUS.G_IO_Modules_Online,
    VI_Reset_Errors := GVL_COMMAND.G_Reset_Errors,
    VI_Emergency_Stop := GVL_STATE.G_Safety_Emergency_Stop,
    VI_System_Mode := GVL_STATE.G_System_Mode,
    VO_Heating_Pump => GVL_STATE.G_DHW_Heating_Pump,
    VO_Circ_Pump => GVL_STATE.G_DHW_Circ_Pump,
    VO_Status => GVL_STATUS.G_DHW_Status
);

// Integrated freeze-hardware diagnostics and maintenance gating
GVL_STATUS.G_Diagnostics.Backup_Pump_Out_Of_Service := NOT GVL_CONFIG.G_Backup_Circulation_Pump_In_Service;
GVL_STATUS.G_Diagnostics.Electric_Heater_Out_Of_Service := NOT GVL_CONFIG.G_Electric_Heater_In_Service;
IF NOT GVL_CONFIG.G_Backup_Circulation_Pump_In_Service THEN
    GVL_STATE.G_Backup_Circulation_Pump := FALSE;
END_IF;
IF NOT GVL_CONFIG.G_Electric_Heater_In_Service THEN
    GVL_STATE.G_Electric_Heater_Enable := FALSE;
END_IF;

GVL_STATE.G_Freeze_Hardware_Degraded := GVL_STATUS.G_Diagnostics.Backup_Pump_Fault OR GVL_STATUS.G_Diagnostics.Electric_Heater_Fault;
GVL_STATE.G_Freeze_Hardware_Failed := GVL_STATUS.G_Diagnostics.Backup_Pump_Fault AND GVL_STATUS.G_Diagnostics.Electric_Heater_Fault;

IF GVL_STATE.G_Freeze_Hardware_Failed THEN
    GVL_STATE.G_Backup_Circulation_Pump := FALSE;
    GVL_STATE.G_Electric_Heater_Enable := FALSE;
    GVL_STATE.G_Safety_Freeze_Risk := TRUE;
END_IF;

FOR L_i := 1 TO GVL_CONSTANTS.C_MAX_MANIFOLDS DO
    GVL_STATUS.G_Diagnostics.Manifold_Pump_Out_Of_Service[L_i] := NOT GVL_CONFIG.G_Manifold_Pump_In_Service[L_i];
    IF NOT GVL_CONFIG.G_Manifold_Pump_In_Service[L_i] THEN
        GVL_STATE.G_Manifold_Pumps[L_i] := FALSE;
    END_IF;
END_FOR;
GVL_STATUS.G_Diagnostics.DHW_Heating_Pump_Out_Of_Service := NOT GVL_CONFIG.G_DHW_Heating_Pump_In_Service;
IF NOT GVL_CONFIG.G_DHW_Heating_Pump_In_Service THEN
    GVL_STATE.G_DHW_Heating_Pump := FALSE;
END_IF;
GVL_STATUS.G_Diagnostics.DHW_Circ_Pump_Out_Of_Service := NOT GVL_CONFIG.G_DHW_Circ_Pump_In_Service;
IF NOT GVL_CONFIG.G_DHW_Circ_Pump_In_Service THEN
    GVL_STATE.G_DHW_Circ_Pump := FALSE;
END_IF;
// >>> BULK_SYNC_ANCHOR: PRG_Heating <<<

// HEATING ADAPTER COPY OUT
FOR L_i := 1 TO 8 DO
    GVL_STATE.G_Zone_Valves[L_i] := L_Zone_Valves_8[L_i];
END_FOR;

(* ---- PRG_IO_Write.st ---- *)
PROGRAM PRG_IO_Write
VAR
    L_i : INT;
END_VAR

// 2. ЗАПИСЬ ВЫХОДОВ (GVL_STATE -> GVL_IO)

// 2.1. Отопление (Термоэлектрические приводы)
FOR L_i := 1 TO 8 DO
    GVL_IO.DO_Zone_Valves[L_i] := GVL_STATE.G_Zone_Valves[L_i];
END_FOR;

// 2.2. Коллекторы (Насосы и смесительные клапаны)
FOR L_i := 1 TO GVL_CONSTANTS.C_MAX_MANIFOLDS DO
    GVL_IO.DO_Manifold_Pumps[L_i] := GVL_STATE.G_Manifold_Pumps[L_i];
    // Масштабирование 0.0-1.0 в 0-1000 для аналогового выхода (0-10В)
    GVL_IO.AO_Manifold_Valves[L_i] := REAL_TO_UINT(GVL_STATE.G_Manifold_Valves[L_i] * 1000.0);
END_FOR;

// 2.4. Вентиляция
FOR L_i := 1 TO GVL_CONSTANTS.C_MAX_SUPPLY_FANS DO
    GVL_IO.AO_Supply_Fans[L_i] := REAL_TO_UINT(GVL_STATE.G_Supply_Fans[L_i] * 100.0);
END_FOR;
FOR L_i := 1 TO GVL_CONSTANTS.C_MAX_EXHAUST_FANS DO
    GVL_IO.AO_Exhaust_Fans[L_i] := REAL_TO_UINT(GVL_STATE.G_Exhaust_Fans[L_i] * 100.0);
END_FOR;

// 2.5. ГВС
GVL_IO.DO_DHW_Heating_Pump := GVL_STATE.G_DHW_Heating_Pump;
GVL_IO.DO_DHW_Circ_Pump := GVL_STATE.G_DHW_Circ_Pump;
IF GVL_STATUS.G_Is_Active_PLC THEN
    GVL_IO.DO_Backup_Circulation_Pump := GVL_STATE.G_Backup_Circulation_Pump;
    GVL_IO.DO_Electric_Heater_Enable := GVL_STATE.G_Electric_Heater_Enable;
ELSE
    GVL_IO.DO_Backup_Circulation_Pump := FALSE;
    GVL_IO.DO_Electric_Heater_Enable := FALSE;
END_IF;

// 2.6. Освещение и шторы (полноценная выдача в физические каналы 0-10В)
FOR L_i := 1 TO 8 DO
    GVL_IO.AO_Lighting_Levels[L_i] := BYTE_TO_UINT(GVL_STATE.G_Lighting_Levels[L_i]) * 10;
END_FOR;
FOR L_i := 1 TO GVL_CONSTANTS.C_MAX_BLINDS DO
    GVL_IO.AO_Blinds_Positions[L_i] := BYTE_TO_UINT(GVL_STATE.G_Blinds_Positions[L_i]) * 10;
END_FOR;

// 2.7. Аварийные выходы (Сирены и клапаны)
IF GVL_ALARM.G_Gas_Fire_Siren AND GVL_ALARM.G_Gas_Alarm_Active THEN
    GVL_IO.DO_Gas_Siren := TRUE;
ELSE
    GVL_IO.DO_Gas_Siren := FALSE;
END_IF;

IF GVL_ALARM.G_Gas_Fire_Siren AND GVL_ALARM.G_Fire_Alarm_Active THEN
    GVL_IO.DO_Fire_Siren := TRUE;
ELSE
    GVL_IO.DO_Fire_Siren := FALSE;
END_IF;

IF GVL_ALARM.G_Security_Siren THEN
    GVL_IO.DO_Security_Siren := TRUE;
ELSE
    GVL_IO.DO_Security_Siren := FALSE;
END_IF;

IF GVL_COMMAND.G_Close_Valve_35 THEN
    GVL_IO.DO_Water_Valve_35_Close := TRUE;
ELSE
    GVL_IO.DO_Water_Valve_35_Close := FALSE;
END_IF;

IF GVL_COMMAND.G_Close_Valve_36 THEN
    GVL_IO.DO_Water_Valve_36_Close := TRUE;
ELSE
    GVL_IO.DO_Water_Valve_36_Close := FALSE;
END_IF;

IF GVL_COMMAND.G_Gas_Valve_Close THEN
    GVL_IO.DO_Gas_Valve_Close := TRUE;
ELSE
    GVL_IO.DO_Gas_Valve_Close := FALSE;
END_IF;

// 2.8. Управление доступом (Периметральная автоматика)
GVL_IO.DO_Gate_Open := GVL_COMMAND.G_Gate_Open;
GVL_IO.DO_Wicket_Open := GVL_COMMAND.G_Wicket_Open;
GVL_IO.DO_Lock_1_Open := GVL_COMMAND.G_Lock_1_Open;
GVL_IO.DO_Lock_1_Close := GVL_COMMAND.G_Lock_1_Close;
GVL_IO.DO_Lock_2_Open := GVL_COMMAND.G_Lock_2_Open;
GVL_IO.DO_Lock_2_Close := GVL_COMMAND.G_Lock_2_Close;

// 2.9. Розетки
GVL_IO.DO_Sockets := GVL_STATE.G_Socket_States;

// Selective zonal water recovery outputs
FOR L_i := 1 TO 32 DO
    GVL_IO.DO_Water_Zone_Enable[L_i] := GVL_STATE.G_Water_Zone_Enable[L_i];
END_FOR;
// >>> BULK_SYNC_ANCHOR: PRG_IO_Write <<<
